Fanuc KAREL source: kt00494.KL

-- PROVISIONAL review KL for V940-1; original PC SHA256 2927928654894c97128c72dadb803d0a5f859ac7bd1ef1d6ec9e5561f602f1f9
-- Incomplete behavior may be omitted. Consult companion uncertainty JSON. Do not deploy.
PROGRAM KT00494
%NOLOCKGROUP
-- UNRESOLVED_DECL P1 type=000102
-- UNRESOLVED_DECL P2 type=000101
-- UNRESOLVED_DECL OUT type=000101
BEGIN
  -- V9_ZERO_TABLE_METADATA_HINT layout=0001; no indexed target words; source/name/runtime held
  -- UNRESOLVED_PC offsets 5-20; opcodes 2E,22,32,35
  -- UNRESOLVED_PC offsets 25-54; opcodes 49,7E,49,60,4A
  -- UNRESOLVED_PC offsets 59-63; opcodes 7F
END KT00494
